INTERFACE I_Patlite

PROPERTY bBuzzerStop : BOOL
SET
END_SET
END_PROPERTY

PROPERTY bStartupBuzzer : BOOL
SET
END_SET
END_PROPERTY

PROPERTY eMachineState : E_MachineState
SET
END_SET
END_PROPERTY

END_INTERFACE

(* stored: Version 1.1.0.1, ProductVersion 3.1.4026.13
   Itf I_Patlite: Id {8503a6b5-cfb3-4e34-822b-289fe1aa92eb}
   Property bBuzzerStop: Id {debee066-b477-418b-8539-daba95734d85}
   Set Set: Id {1a1894ce-67b4-42a8-866f-3f50341604eb}
   Property bStartupBuzzer: Id {6ea3a3d8-41c0-4e95-93e6-9d603328cdeb}
   Set Set: Id {9be3250a-9098-4865-b2fe-8b923ef239d3}
   Property eMachineState: Id {6420d867-462d-4471-98d3-951b3d1ec600}
   Set Set: Id {707c826a-b2b1-4cc7-9e79-2bfe47087be7} *)
